FUNCTION_BLOCK FB_Calcul_Position_V4
VAR_INPUT

	lrPosCodeurDroite	: LREAL;
	lrPosCodeurGauche	: LREAL;
	lrEntraxeCodeur		: LREAL;

	boSetPosInitiale	: BOOL;
	lrPosInitialeX		: LREAL;
	lrPosInitialeY		: LREAL;
	lrPosInitialeAngle	: LREAL;	// en [°], le 0° vers Y+, sens horaire

END_VAR
VAR_OUTPUT
	
	lrPosActuelleX		: LREAL;
	lrPosActuelleY		: LREAL;
	lrPosActuelleAngle	: LREAL;

END_VAR
VAR
	
	lrPosCodeurDroiteDernierCycle	: LREAL;
	lrPosCodeurGaucheDernierCycle	: LREAL;
	lrPosActuelleAngleRadian		: LREAL;	

	lrDeltaCodeurDroite		: LREAL;
	lrDeltaCodeurGauche		: LREAL;
	
	lrDeltaDistance		: LREAL;
	lrDeltaAngle		: lreal;
	
END_VAR
VAR CONSTANT
	
	lrValeurPi	: LREAL := 3.1415926535897932384626433832795;

END_VAR

//Gestion set pos initiale

IF boSetPosInitiale THEN
	
	lrPosActuelleX := lrPosInitialeX;
	lrPosActuelleY := lrPosInitialeY;
	lrPosActuelleAngle := lrPosInitialeAngle;
	lrPosActuelleAngleRadian := lrPosInitialeAngle * ( lrValeurPi / 180 );
	
	lrPosCodeurDroiteDernierCycle := lrPosCodeurDroite;
	lrPosCodeurGaucheDernierCycle := lrPosCodeurGauche;

END_IF

//Calcul des deltas codeurs

lrDeltaCodeurDroite := lrPosCodeurDroite - lrPosCodeurDroiteDernierCycle;
lrDeltaCodeurGauche := lrPosCodeurGauche - lrPosCodeurGaucheDernierCycle;

//Calcul distance moyenne et angle

lrDeltaDistance	:= ( lrDeltaCodeurDroite + lrDeltaCodeurGauche ) / 2;
lrDeltaAngle	:= ATAN ( ( lrDeltaCodeurGauche - lrDeltaCodeurDroite ) / lrEntraxeCodeur );

//Calcul pos du robot

lrPosActuelleX := lrPosActuelleX + ( lrDeltaDistance * SIN ( lrPosActuelleAngleRadian ) );
lrPosActuelleY := lrPosActuelleY + ( lrDeltaDistance * COS ( lrPosActuelleAngleRadian ) );

lrPosActuelleAngleRadian := lrPosActuelleAngleRadian + lrDeltaAngle;

IF lrPosActuelleAngleRadian < 0 THEN
	
	lrPosActuelleAngleRadian := lrPosActuelleAngleRadian + ( 2.0 * lrValeurPi );
	
ELSIF lrPosActuelleAngleRadian >= ( 2 * lrValeurPi ) THEN
	
	lrPosActuelleAngleRadian := lrPosActuelleAngleRadian - ( 2.0 * lrValeurPi );

END_IF

lrPosActuelleAngle := lrPosActuelleAngleRadian * ( 180 / lrValeurPi );

lrPosCodeurDroiteDernierCycle := lrPosCodeurDroite;
lrPosCodeurGaucheDernierCycle := lrPosCodeurGauche;

END_FUNCTION_BLOCK

(* stored: Version 1.1.0.1, ProductVersion 3.1.4022.18
   POU FB_Calcul_Position_V4: Id {02018b14-d3ab-4111-b46b-8646e09a38fe}, SpecialFunc None *)
